// TIA Portal V18 export
// export: Created 2026-01-09T11:32:04.6391025Z, ExportSetting WithDefaults, DisplayName Totally Integrated Automation Portal, DisplayVersion V18 Update 5, DisplayName TIA Portal Openness, DisplayVersion V18 Update 5, DisplayName TIA Portal Teamcenter Gateway, DisplayVersion V18, DisplayName TIA Portal Version Control Interface, DisplayVersion V18, DisplayName SINAMICS Startdrive Advanced, DisplayVersion V18 SP2 Update 1, DisplayName SINAMICS Startdrive G110M, G120, G120C, G120D, G120P, G115D, DisplayVersion V18 SP2 Update 1, DisplayName SINAMICS Startdrive G130, G150, S120, S150, SINAMICS MV, S210, G220, S200, DisplayVersion V18 SP2 Update 1, DisplayName STEP 7 Professional, DisplayVersion V18 Update 5, DisplayName STEP 7 Safety, DisplayVersion V18, DisplayName WinCC Professional, DisplayVersion V18 Update 5
TagTable "PM_CycleTime"
  PM_TotalCycleTimeNo[13] : Real  (%DB[PM_CountCycleDBNum].DBD[PM_TotalCycleT13Address], CPU S71500-2PN_TP700, 1 s)
  PM_TotalCycleTimeNo[17] : Real  (%DB[PM_CountCycleDBNum].DBD[PM_TotalCycleT17Address], CPU S71500-2PN_TP700, 1 s)
  PM_TotalCycleTimeNo[11] : Real  (%DB[PM_CountCycleDBNum].DBD[PM_TotalCycleT11Address], CPU S71500-2PN_TP700, 1 s)
  PM_TotalCycleTimeNo[20] : Real  (%DB[PM_CountCycleDBNum].DBD[PM_TotalCycleT20Address], CPU S71500-2PN_TP700, 1 s)
  PM_TotalCycleTimeNo[04] : Real  (%DB[PM_CountCycleDBNum].DBD[PM_TotalCycleT04Address], CPU S71500-2PN_TP700, 1 s)
  PM_TotalCycleTimeNo[10] : Real  (%DB[PM_CountCycleDBNum].DBD[PM_TotalCycleT10Address], CPU S71500-2PN_TP700, 1 s)
  PM_TotalCycleTimeNo[06] : Real  (%DB[PM_CountCycleDBNum].DBD[PM_TotalCycleT06Address], CPU S71500-2PN_TP700, 1 s)
  PM_TotalCycleTimeNo[15] : Real  (%DB[PM_CountCycleDBNum].DBD[PM_TotalCycleT15Address], CPU S71500-2PN_TP700, 1 s)
  PM_TotalCycleTimeNo[01] : Real  (%DB[PM_CountCycleDBNum].DBD[PM_TotalCycleT01Address], CPU S71500-2PN_TP700, 1 s)
  PM_TotalCycleTimeNo[14] : Real  (%DB[PM_CountCycleDBNum].DBD[PM_TotalCycleT14Address], CPU S71500-2PN_TP700, 1 s)
  PM_TotalCycleTimeNo[16] : Real  (%DB[PM_CountCycleDBNum].DBD[PM_TotalCycleT16Address], CPU S71500-2PN_TP700, 1 s)
  PM_TotalCycleTimeNo[0] : Real  (%DB[PM_CountCycleDBNum].DBD[PM_TotalCycleT0Address], CPU S71500-2PN_TP700, 1 s)
  PM_TotalCycleTimeNo[02] : Real  (%DB[PM_CountCycleDBNum].DBD[PM_TotalCycleT02Address], CPU S71500-2PN_TP700, 1 s)
  PM_TotalCycleTimeNo[07] : Real  (%DB[PM_CountCycleDBNum].DBD[PM_TotalCycleT07Address], CPU S71500-2PN_TP700, 1 s)
  PM_TotalCycleTimeNo[05] : Real  (%DB[PM_CountCycleDBNum].DBD[PM_TotalCycleT05Address], CPU S71500-2PN_TP700, 1 s)
  PM_TotalCycleTimeNo[09] : Real  (%DB[PM_CountCycleDBNum].DBD[PM_TotalCycleT09Address], CPU S71500-2PN_TP700, 1 s)
  PM_TotalCycleTimeNo[21] : Real  (%DB[PM_CountCycleDBNum].DBD[PM_TotalCycleT21Address], CPU S71500-2PN_TP700, 1 s)
  PM_TotalCycleTimeNo[19] : Real  (%DB[PM_CountCycleDBNum].DBD[PM_TotalCycleT19Address], CPU S71500-2PN_TP700, 1 s)
  PM_TotalCycleTimeNo[12] : Real  (%DB[PM_CountCycleDBNum].DBD[PM_TotalCycleT12Address], CPU S71500-2PN_TP700, 1 s)
  PM_TotalCycleTimeNo[03] : Real  (%DB[PM_CountCycleDBNum].DBD[PM_TotalCycleT03Address], CPU S71500-2PN_TP700, 1 s)
  PM_TotalCycleTimeNo[08] : Real  (%DB[PM_CountCycleDBNum].DBD[PM_TotalCycleT08Address], CPU S71500-2PN_TP700, 1 s)
  PM_TotalCycleTimeNo[18] : Real  (%DB[PM_CountCycleDBNum].DBD[PM_TotalCycleT18Address], CPU S71500-2PN_TP700, 1 s)
  PM_MachineCycleTimeNo[0] : Real  (%DB[PM_CountCycleDBNum].DBD[PM_MachCycleT0Address], CPU S71500-2PN_TP700, 1 s)
  PM_MachineCycleTimeNo[01] : Real  (%DB[PM_CountCycleDBNum].DBD[PM_MachCycleT01Address], CPU S71500-2PN_TP700, 1 s)
  PM_MachineCycleTimeNo[10] : Real  (%DB[PM_CountCycleDBNum].DBD[PM_MachCycleT10Address], CPU S71500-2PN_TP700, 1 s)
  PM_MachineCycleTimeNo[11] : Real  (%DB[PM_CountCycleDBNum].DBD[PM_MachCycleT11Address], CPU S71500-2PN_TP700, 1 s)
  PM_MachineCycleTimeNo[12] : Real  (%DB[PM_CountCycleDBNum].DBD[PM_MachCycleT12Address], CPU S71500-2PN_TP700, 1 s)
  PM_MachineCycleTimeNo[13] : Real  (%DB[PM_CountCycleDBNum].DBD[PM_MachCycleT13Address], CPU S71500-2PN_TP700, 1 s)
  PM_MachineCycleTimeNo[14] : Real  (%DB[PM_CountCycleDBNum].DBD[PM_MachCycleT14Address], CPU S71500-2PN_TP700, 1 s)
  PM_MachineCycleTimeNo[15] : Real  (%DB[PM_CountCycleDBNum].DBD[PM_MachCycleT15Address], CPU S71500-2PN_TP700, 1 s)
  PM_MachineCycleTimeNo[16] : Real  (%DB[PM_CountCycleDBNum].DBD[PM_MachCycleT16Address], CPU S71500-2PN_TP700, 1 s)
  PM_MachineCycleTimeNo[17] : Real  (%DB[PM_CountCycleDBNum].DBD[PM_MachCycleT17Address], CPU S71500-2PN_TP700, 1 s)
  PM_MachineCycleTimeNo[18] : Real  (%DB[PM_CountCycleDBNum].DBD[PM_MachCycleT18Address], CPU S71500-2PN_TP700, 1 s)
  PM_MachineCycleTimeNo[19] : Real  (%DB[PM_CountCycleDBNum].DBD[PM_MachCycleT19Address], CPU S71500-2PN_TP700, 1 s)
  PM_MachineCycleTimeNo[02] : Real  (%DB[PM_CountCycleDBNum].DBD[PM_MachCycleT02Address], CPU S71500-2PN_TP700, 1 s)
  PM_MachineCycleTimeNo[20] : Real  (%DB[PM_CountCycleDBNum].DBD[PM_MachCycleT20Address], CPU S71500-2PN_TP700, 1 s)
  PM_MachineCycleTimeNo[21] : Real  (%DB[PM_CountCycleDBNum].DBD[PM_MachCycleT21Address], CPU S71500-2PN_TP700, 1 s)
  PM_MachineCycleTimeNo[03] : Real  (%DB[PM_CountCycleDBNum].DBD[PM_MachCycleT03Address], CPU S71500-2PN_TP700, 1 s)
  PM_MachineCycleTimeNo[04] : Real  (%DB[PM_CountCycleDBNum].DBD[PM_MachCycleT04Address], CPU S71500-2PN_TP700, 1 s)
  PM_MachineCycleTimeNo[05] : Real  (%DB[PM_CountCycleDBNum].DBD[PM_MachCycleT05Address], CPU S71500-2PN_TP700, 1 s)
  PM_MachineCycleTimeNo[06] : Real  (%DB[PM_CountCycleDBNum].DBD[PM_MachCycleT06Address], CPU S71500-2PN_TP700, 1 s)
  PM_MachineCycleTimeNo[07] : Real  (%DB[PM_CountCycleDBNum].DBD[PM_MachCycleT07Address], CPU S71500-2PN_TP700, 1 s)
  PM_MachineCycleTimeNo[08] : Real  (%DB[PM_CountCycleDBNum].DBD[PM_MachCycleT08Address], CPU S71500-2PN_TP700, 1 s)
  PM_MachineCycleTimeNo[09] : Real  (%DB[PM_CountCycleDBNum].DBD[PM_MachCycleT09Address], CPU S71500-2PN_TP700, 1 s)
  PM_MachCycleT0Address : UInt  (1 s)
  PM_MachCycleT01Address : UInt  (1 s)
  PM_MachCycleT02Address : UInt  (1 s)
  PM_MachCycleT03Address : UInt  (1 s)
  PM_MachCycleT04Address : UInt  (1 s)
  PM_MachCycleT05Address : UInt  (1 s)
  PM_MachCycleT06Address : UInt  (1 s)
  PM_MachCycleT07Address : UInt  (1 s)
  PM_MachCycleT08Address : UInt  (1 s)
  PM_MachCycleT09Address : UInt  (1 s)
  PM_MachCycleT10Address : UInt  (1 s)
  PM_MachCycleT11Address : UInt  (1 s)
  PM_MachCycleT12Address : UInt  (1 s)
  PM_MachCycleT13Address : UInt  (1 s)
  PM_MachCycleT14Address : UInt  (1 s)
  PM_MachCycleT15Address : UInt  (1 s)
  PM_MachCycleT16Address : UInt  (1 s)
  PM_MachCycleT17Address : UInt  (1 s)
  PM_MachCycleT18Address : UInt  (1 s)
  PM_MachCycleT19Address : UInt  (1 s)
  PM_MachCycleT20Address : UInt  (1 s)
  PM_MachCycleT21Address : UInt  (1 s)
  PM_TotalCycleT0Address : UInt  (1 s)
  PM_TotalCycleT01Address : UInt  (1 s)
  PM_TotalCycleT02Address : UInt  (1 s)
  PM_TotalCycleT03Address : UInt  (1 s)
  PM_TotalCycleT04Address : UInt  (1 s)
  PM_TotalCycleT05Address : UInt  (1 s)
  PM_TotalCycleT06Address : UInt  (1 s)
  PM_TotalCycleT07Address : UInt  (1 s)
  PM_TotalCycleT08Address : UInt  (1 s)
  PM_TotalCycleT09Address : UInt  (1 s)
  PM_TotalCycleT10Address : UInt  (1 s)
  PM_TotalCycleT11Address : UInt  (1 s)
  PM_TotalCycleT12Address : UInt  (1 s)
  PM_TotalCycleT13Address : UInt  (1 s)
  PM_TotalCycleT14Address : UInt  (1 s)
  PM_TotalCycleT15Address : UInt  (1 s)
  PM_TotalCycleT16Address : UInt  (1 s)
  PM_TotalCycleT17Address : UInt  (1 s)
  PM_TotalCycleT18Address : UInt  (1 s)
  PM_TotalCycleT19Address : UInt  (1 s)
  PM_TotalCycleT20Address : UInt  (1 s)
  PM_TotalCycleT21Address : UInt  (1 s)
